KUKA KRL program: dejar_darsena2.src, dejar_darsena2.dat

--- dejar_darsena2.src ---
&ACCESS RVP1
&REL 1318
&COMMENT Dejada Darsena 2
DEF Dejar_Darsena2()

;*************************************************;
;***          DEJAR PRODUCTO EN EL PALE        ***;
;*                                               *;
;*                 Movimientos.                  *;
;*************************************************;




IF  NOT INIT THEN
 ;FOLD INI
 ;FOLD BASISTECH INI
 GLOBAL INTERRUPT DECL 3 WHEN $STOPMESS==TRUE DO IR_STOPM ( )
 INTERRUPT ON 3
 BAS (#INITMOV,0 )
 ;ENDFOLD (BASISTECH INI)
 ;FOLD GRIPPERTECH INI
 ;USER_GRP (0,DUMMY,DUMMY,GDEFAULT )
 ;ENDFOLD (GRIPPERTECH INI)
 ;FOLD USER INI
 ;Make your modifications here

 ;ENDFOLD (USER INI)
   ;ENDFOLD (INI)
   INIT=TRUE
 ENDIF
continue

;CAMBIO DE BASE-->BASE DARSENA 2
FAPROXIMACION_DEJADA.BASE_NO=1
FDEJADA.BASE_NO=1
FSALIDA_DEJADA.BASE_NO=1



; ;EN DARSENA 2 EL ROBOT CAMBIA EL VALOR DE T
;
;         IF (XDEJADA.X>376) THEN
;               XAPROXIMACION_DEJADA.t=43
;               XDEJADA.t=43
;               XSALIDA_DEJADA.t=43
;
;                       IF  (XDEJADA.A>170) THEN
;                         XAPROXIMACION_DEJADA.t=3
;                         XDEJADA.t=3
;                         XSALIDA_DEJADA.t=3
;                       ENDIF
;
;         ENDIF
;
;
;         IF ( (XDEJADA.X<=376) AND (XDEJADA.X>50) ) THEN
;               XAPROXIMACION_DEJADA.t=42
;               XDEJADA.t=42
;               XSALIDA_DEJADA.t=42
;
;         ENDIF
;
;
;         IF (XDEJADA.X<70)  THEN
;               XAPROXIMACION_DEJADA.t=10
;               XDEJADA.t=10
;               XSALIDA_DEJADA.t=10
;         ENDIF


;IGUALO LA ORIENTCION DE LA ENTRADA A LA DARSENA A LA DEL PTO DE DEJADA
    XENTRADA_DEJADA_DARS2.A=XAPROXIMACION_DEJADA.A
    XENTRADA_DEJADA_DARS2.B=XAPROXIMACION_DEJADA.B
    XENTRADA_DEJADA_DARS2.C=XAPROXIMACION_DEJADA.C
    XENTRADA_DEJADA_DARS2.t=XAPROXIMACION_DEJADA.t


;LA ORI EN DARSENA DOS, TIENE LA Z NEGATIVA, CORREGIMOS EL SIGNO DE LA DEJADA

    XAPROXIMACION_DEJADA.Z=-XAPROXIMACION_DEJADA.Z
    XDEJADA.Z=-XDEJADA.Z
    XSALIDA_DEJADA.Z=-XSALIDA_DEJADA.Z


;FOLD PTP ENTRADA_DEJADA_DAR2 CONT Vel=100 % PDAT127 Tool[2]:MORDAZA Base[1]:DARSENA2;%{PE}%R 5.6.16,%MKUKATPBASIS,%CMOVE,%VPTP,%P 1:PTP, 2:ENTRADA_DEJADA_DAR2, 3:C_PTP, 5:100, 7:PDAT127
$BWDSTART=FALSE
PDAT_ACT=PPDAT127
FDAT_ACT=FENTRADA_DEJADA_DAR2
BAS(#PTP_PARAMS,100)
PTP XENTRADA_DEJADA_DAR2 C_PTP
;ENDFOLD


;FOLD PTP APROXIMACION_DEJADA Vel=100 % PDAT129 Tool[0] Base[0];%{PE}%R 8.3.22,%MKUKATPBASIS,%CMOVE,%VPTP,%P 1:PTP, 2:aPROXIMACION_DEJADA, 3:, 5:100, 7:PDAT129
$BWDSTART=FALSE
PDAT_ACT=PPDAT1
FDAT_ACT=FAPROXIMACION_DEJADA
BAS(#PTP_PARAMS,100)
PTP xAproximacion_dejada C_PTP
;ENDFOLD


TRIGGER WHEN DISTANCE = 1 DELAY=-100 DO PULSE(ABRIR_GARRAS,TRUE,0.1)

;FOLD LIN DEJADA  Vel=2 m/s CPDAT46 Tool[0] Base[0];%{PE}%R 8.3.22,%MKUKATPBASIS,%CMOVE,%VLIN,%P 1:LIN, 2:DEJADA, 3:, 5:2, 7:CPDAT46
$BWDSTART=FALSE
LDAT_ACT=LCPDAT1
FDAT_ACT=FDEJADA
BAS(#CP_PARAMS,2)
LIN XDEJADA C_DIS
;ENDFOLD

EXTENDER_PISADORES=FALSE

WAIT FOR (GARRAS_ABIERTAS)


TRIGGER WHEN DISTANCE = 1 DELAY=-100 DO PULSE(CERRAR_GARRAS,TRUE,0.1)

;FOLD LIN Salida_DEJADA Vel=2 m/s CPDAT46 Tool[0] Base[0];%{PE}%R 8.3.22,%MKUKATPBASIS,%CMOVE,%VLIN,%P 1:LIN, 2:DEJADA, 3:, 5:2, 7:CPDAT46
$BWDSTART=FALSE
LDAT_ACT=LCPDAT1
FDAT_ACT=FSalida_DEJADA
BAS(#CP_PARAMS,2)
LIN XSalida_DEJADA C_DIS
;ENDFOLD


;FOLD PTP ENTRADA_DEJADA_DAR2 CONT Vel=100 % PDAT128 Tool[2]:MORDAZA Base[1]:DARSENA2;%{PE}%R 5.6.16,%MKUKATPBASIS,%CMOVE,%VPTP,%P 1:PTP, 2:ENTRADA_DEJADA_DAR2, 3:C_PTP, 5:100, 7:PDAT128
$BWDSTART=FALSE
PDAT_ACT=PPDAT1
FDAT_ACT=FENTRADA_DEJADA_DAR2
BAS(#PTP_PARAMS,100)
PTP XENTRADA_DEJADA_DAR2 C_PTP
;ENDFOLD


CONTADOR_SACOS_DARSENA2=CONTADOR_SACOS_DARSENA2+1

;FOLD PTP home Vel=100 % PDAT130;%{PE}%R 5.6.16,%MKUKATPBASIS,%CMOVE,%VPTP,%P 1:PTP, 2:home, 3:, 5:100, 7:PDAT130
$BWDSTART=FALSE
PDAT_ACT=PPDAT1
FDAT_ACT=Fhome
BAS(#PTP_PARAMS,100)
$H_POS=XHOME
PTP Xhome
;ENDFOLD

END

--- dejar_darsena2.dat ---
&ACCESS RVP1
&REL 1318
&COMMENT Dejada Darsena 2
DEFDAT  DEJAR_DARSENA2 PUBLIC

;FOLD EXTERNAL DECLARATIONS;%{PE}%MKUKATPBASIS,%CEXT,%VCOMMON,%P
;FOLD BASISTECH EXT;%{PE}%MKUKATPBASIS,%CEXT,%VEXT,%P
EXT  BAS (BAS_COMMAND  :IN,REAL  :IN )
DECL INT SUCCESS
;ENDFOLD (BASISTECH EXT)
;FOLD USER EXT;%{E}%MKUKATPUSER,%CEXT,%VEXT,%P
;Make here your modifications

;ENDFOLD (USER EXT)
;ENDFOLD (EXTERNAL DECLARATIONS)

DECL BASIS_SUGG_T LAST_BASIS={POINT1[] "DEJADA                  ",POINT2[] "DEJADA                  ",CP_PARAMS[] "CPDAT46                 ",PTP_PARAMS[] "PDAT129                 ",CONT[] "                        ",CP_VEL[] "2                       ",PTP_VEL[] "100                     ",SYNC_PARAMS[] "SYNCDAT                 ",SPL_NAME[] "S0                      "}
; DATOS


DECL PDAT PPDAT1={VEL 100.0,ACC 100.0,APO_DIST 100.0}


DECL E6POS XENTRADA_DEJADA_DAR2={X 279.762207,Y 309.286407,Z -1850.89099,A 176.867798,B 0.237935707,C 0.131209806,S 6,T 58,E1 0.0,E2 0.0,E3 0.0,E4 0.0,E5 0.0,E6 0.0}
DECL FDAT FENTRADA_DEJADA_DAR2={TOOL_NO 2,BASE_NO 1,IPO_FRAME #BASE,POINT2[] " ",TQ_STATE FALSE}


DECL LDAT LCPDAT1={VEL 2.0,ACC 100.0,APO_DIST 100.0,APO_FAC 50.0,ORI_TYP #VAR,CIRC_TYP #BASE,JERK_FAC 50.0,EXAX_IGN 0}

DECL PDAT PPDAT128={VEL 100.0,ACC 100.0,APO_DIST 100.0,APO_MODE #CPTP}
DECL E6POS XENTRADA_DEJADA_DAR3={X 465.442902,Y 717.486328,Z -1811.01501,A -3.48240089,B -0.0301607605,C 0.0118598901,S 2,T 43,E1 0.0,E2 0.0,E3 0.0,E4 0.0,E5 0.0,E6 0.0}
DECL FDAT FENTRADA_DEJADA_DAR3={TOOL_NO 2,BASE_NO 3,IPO_FRAME #BASE,POINT2[] " ",TQ_STATE FALSE}
DECL FDAT FENTRADA_DEJADA_DARS1={TOOL_NO 2,BASE_NO 4,IPO_FRAME #BASE,POINT2[] " ",TQ_STATE FALSE}
DECL E6POS XENTRADA_DEJADA_DARS1={X 403.819214,Y 727.108398,Z 1797.81494,A 90.0,B 0.0,C 180.0,S 2,T 42,E1 0.0,E2 0.0,E3 0.0,E4 0.0,E5 0.0,E6 0.0}


DECL PDAT PPDAT127={VEL 100.0,ACC 100.0,APO_DIST 100.0,APO_MODE #CPTP}
ENDDAT
